PROGRAM A08_CodeInfoCtrl
VAR

	fbClearPackCodeInfo			:	FB_CODE_ClearCodeInfo;
	fbClearIntermediateCodeInfo		:	FB_CODE_ClearCodeInfo;
	fbClearOuerCodeInfo			:	FB_CODE_ClearCodeInfo;
	fbClearCaseCodeInfo			:	FB_CODE_ClearCodeInfo;

	fbGS1ClearPackCodeInfo			:	FB_GS1_ClearCodeInfo;

	sFullCode	:STRING := '1234567890ABCDEFGFQQQQ';
	sGetItem : STRING;
	eGS1_AIType		: 	E_GS1_CodeAIType;

	fbValidateExplicitCode: FB_GS1_ValidateExplicitCode;
	bValidationOK : BOOL;

	fbBATOuterSerializator	: FB_CODE_BATSerializator;

	sSerialCode1: STRING(25);
	bGenereteCode		: BOOL;
	nSecquentionalCounter2		: UDINT;
	bFNC1Add		: BOOL;

	bDone		: BOOL;
	bIthemtype 	: BOOL;

	sSerialCode2: STRING(25);
	nSecquentionalCounter1		: UDINT;
	bFNC1Add1		: BOOL;

	fbBATOuterCodeGenerator		: FB_CODE_OuterCodeGenerator;

	bGenereteCode3	: BOOL;
	nNumberOfCodeGenrerated	: INT;
	nSecquentionalCounter3		: UDINT;
	aCodePrinterBuffer		: ARRAY[1..25] OF T_OUTER_Barcode;
		bDone2		: BOOL;


END_VAR

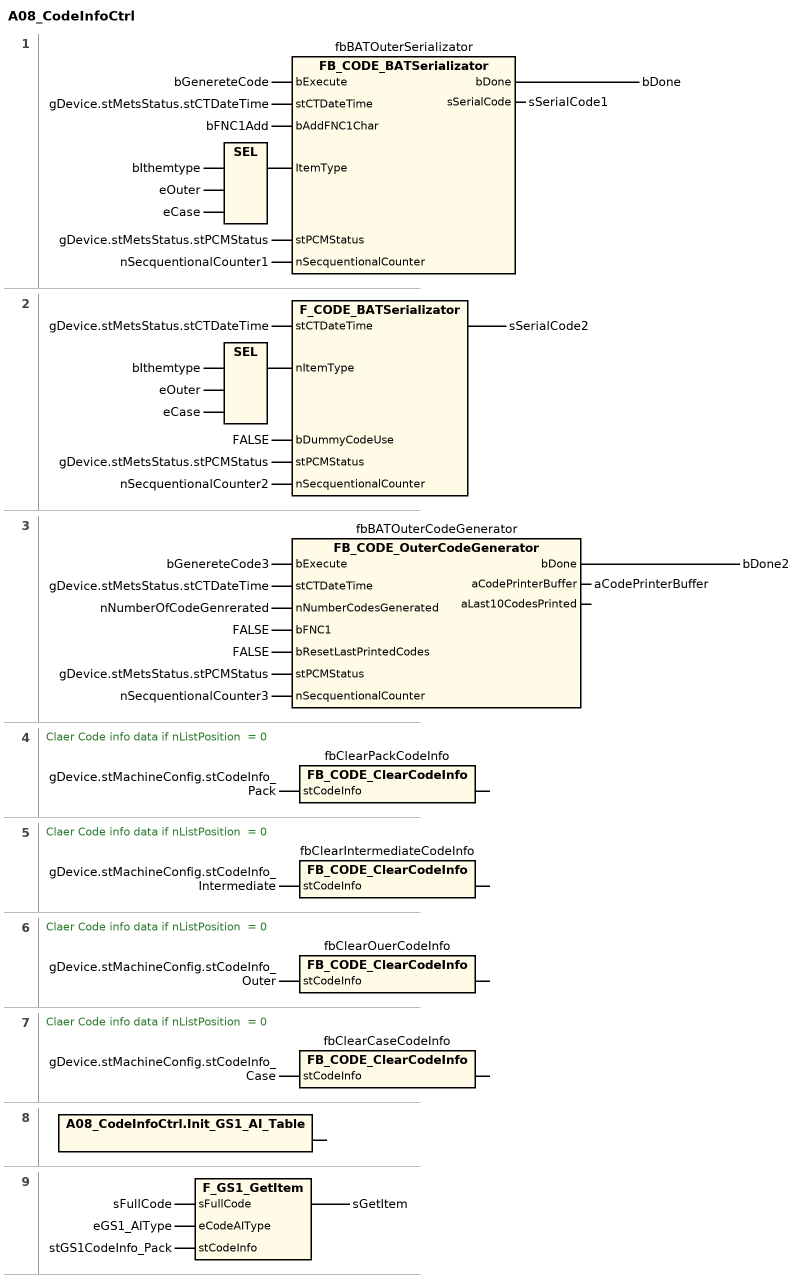
// NETWORK 1
fbBATOuterSerializator(
    bExecute := bGenereteCode,
    stCTDateTime := gDevice.stMetsStatus.stCTDateTime,
    bAddFNC1Char := bFNC1Add,
    ItemType := SEL(bIthemtype, eOuter, eCase),
    stPCMStatus := gDevice.stMetsStatus.stPCMStatus,
    nSecquentionalCounter := nSecquentionalCounter1,
    sSerialCode => sSerialCode1); // FB_CODE_BATSerializator
bDone := fbBATOuterSerializator.bDone;

// NETWORK 2
sSerialCode2 := F_CODE_BATSerializator(stCTDateTime := gDevice.stMetsStatus.stCTDateTime, nItemType := SEL(bIthemtype, eOuter, eCase), bDummyCodeUse := FALSE, stPCMStatus := gDevice.stMetsStatus.stPCMStatus, nSecquentionalCounter := nSecquentionalCounter2);

// NETWORK 3
fbBATOuterCodeGenerator(
    bExecute := bGenereteCode3,
    stCTDateTime := gDevice.stMetsStatus.stCTDateTime,
    nNumberCodesGenerated := nNumberOfCodeGenrerated,
    bFNC1 := FALSE,
    bResetLastPrintedCodes := FALSE,
    stPCMStatus := gDevice.stMetsStatus.stPCMStatus,
    nSecquentionalCounter := nSecquentionalCounter3,
    aCodePrinterBuffer => aCodePrinterBuffer); // FB_CODE_OuterCodeGenerator
bDone2 := fbBATOuterCodeGenerator.bDone;

// NETWORK 4
//  Claer Code info data if nListPosition  = 0
fbClearPackCodeInfo(stCodeInfo := gDevice.stMachineConfig.stCodeInfo_Pack); // FB_CODE_ClearCodeInfo

// NETWORK 5
// Claer Code info data if nListPosition  = 0
fbClearIntermediateCodeInfo(stCodeInfo := gDevice.stMachineConfig.stCodeInfo_Intermediate); // FB_CODE_ClearCodeInfo

// NETWORK 6
// Claer Code info data if nListPosition  = 0
fbClearOuerCodeInfo(stCodeInfo := gDevice.stMachineConfig.stCodeInfo_Outer); // FB_CODE_ClearCodeInfo

// NETWORK 7
// Claer Code info data if nListPosition  = 0
fbClearCaseCodeInfo(stCodeInfo := gDevice.stMachineConfig.stCodeInfo_Case); // FB_CODE_ClearCodeInfo

// NETWORK 8
A08_CodeInfoCtrl.Init_GS1_AI_Table();

// NETWORK 9
sGetItem := F_GS1_GetItem(sFullCode := sFullCode, eCodeAIType := eGS1_AIType, stCodeInfo := stGS1CodeInfo_Pack);

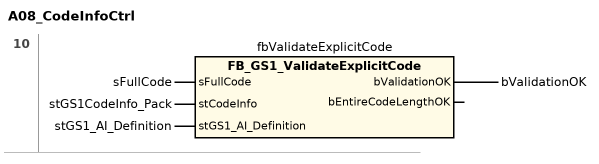
// NETWORK 10
fbValidateExplicitCode(
    sFullCode := sFullCode,
    stCodeInfo := stGS1CodeInfo_Pack,
    stGS1_AI_Definition := stGS1_AI_Definition); // FB_GS1_ValidateExplicitCode
bValidationOK := fbValidateExplicitCode.bValidationOK;

ACTION Init_GS1_AI_Table:
aGS1_Decode_AI[1].sAI_Id	:= stGS1_AI_Definition.stAI_01_Lvl1.sAI_Id;
aGS1_Decode_AI[1].bFixed	:= stGS1_AI_Definition.stAI_01_Lvl1.bFixed;
aGS1_Decode_AI[1].nLength	:= stGS1_AI_Definition.stAI_01_Lvl1.nLength;

aGS1_Decode_AI[2].sAI_Id	:= stGS1_AI_Definition.stAI_10.sAI_Id;
aGS1_Decode_AI[2].bFixed	:= stGS1_AI_Definition.stAI_10.bFixed;
aGS1_Decode_AI[2].nLength	:= stGS1_AI_Definition.stAI_10.nLength;

aGS1_Decode_AI[3].sAI_Id	:= stGS1_AI_Definition.stAI_11.sAI_Id;
aGS1_Decode_AI[3].bFixed	:= stGS1_AI_Definition.stAI_11.bFixed;
aGS1_Decode_AI[3].nLength	:= stGS1_AI_Definition.stAI_11.nLength;

aGS1_Decode_AI[4].sAI_Id	:= stGS1_AI_Definition.stAI_15.sAI_Id;
aGS1_Decode_AI[4].bFixed	:= stGS1_AI_Definition.stAI_15.bFixed;
aGS1_Decode_AI[4].nLength	:= stGS1_AI_Definition.stAI_15.nLength;

aGS1_Decode_AI[5].sAI_Id	:= stGS1_AI_Definition.stAI_17.sAI_Id;
aGS1_Decode_AI[5].bFixed	:= stGS1_AI_Definition.stAI_17.bFixed;
aGS1_Decode_AI[5].nLength	:= stGS1_AI_Definition.stAI_17.nLength;

aGS1_Decode_AI[6].sAI_Id	:= stGS1_AI_Definition.stAI_21.sAI_Id;
aGS1_Decode_AI[6].bFixed	:= stGS1_AI_Definition.stAI_21.bFixed;
aGS1_Decode_AI[6].nLength	:= stGS1_AI_Definition.stAI_21.nLength;

aGS1_Decode_AI[7].sAI_Id	:= stGS1_AI_Definition.stAI_240.sAI_Id;
aGS1_Decode_AI[7].bFixed	:= stGS1_AI_Definition.stAI_240.bFixed;
aGS1_Decode_AI[7].nLength	:= stGS1_AI_Definition.stAI_240.nLength;

aGS1_Decode_AI[8].sAI_Id	:= stGS1_AI_Definition.stAI_8005.sAI_Id;
aGS1_Decode_AI[8].bFixed	:= stGS1_AI_Definition.stAI_8005.bFixed;
aGS1_Decode_AI[8].nLength	:= stGS1_AI_Definition.stAI_8005.nLength;

aGS1_Decode_AI[9].sAI_Id	:= stGS1_AI_Definition.stAI_8006.sAI_Id;
aGS1_Decode_AI[9].bFixed	:= stGS1_AI_Definition.stAI_8006.bFixed;
aGS1_Decode_AI[9].nLength	:= stGS1_AI_Definition.stAI_8006.nLength;

aGS1_Decode_AI[10].sAI_Id	:= stGS1_AI_Definition.stAI_8008.sAI_Id;
aGS1_Decode_AI[10].bFixed	:= stGS1_AI_Definition.stAI_8008.bFixed;
aGS1_Decode_AI[10].nLength	:= stGS1_AI_Definition.stAI_8008.nLength;

aGS1_Decode_AI[11].sAI_Id	:= stGS1_AI_Definition.stAI_91.sAI_Id;
aGS1_Decode_AI[11].bFixed	:= stGS1_AI_Definition.stAI_91.bFixed;
aGS1_Decode_AI[11].nLength	:= stGS1_AI_Definition.stAI_91.nLength;

aGS1_Decode_AI[12].sAI_Id	:= stGS1_AI_Definition.stAI_92.sAI_Id;
aGS1_Decode_AI[12].bFixed	:= stGS1_AI_Definition.stAI_92.bFixed;
aGS1_Decode_AI[12].nLength	:= stGS1_AI_Definition.stAI_92.nLength;

aGS1_Decode_AI[13].sAI_Id	:= stGS1_AI_Definition.stAI_93.sAI_Id;
aGS1_Decode_AI[13].bFixed	:= stGS1_AI_Definition.stAI_93.bFixed;
aGS1_Decode_AI[13].nLength	:= stGS1_AI_Definition.stAI_93.nLength;

aGS1_Decode_AI[14].sAI_Id	:= stGS1_AI_Definition.stAI_94.sAI_Id;
aGS1_Decode_AI[14].bFixed	:= stGS1_AI_Definition.stAI_94.bFixed;
aGS1_Decode_AI[14].nLength	:= stGS1_AI_Definition.stAI_94.nLength;
END_ACTION

END_PROGRAM

(* stored: Version 1.1.0.1
   POU A08_CodeInfoCtrl: Id {29060727-3d7a-4435-a8f5-e1534cf8ade8}, SpecialFunc None
   Action Init_GS1_AI_Table: Id {ce778151-ebfe-4084-983c-23b628c9080f} *)
